FUNCTION F_VoltageToCurrentConvert : REAL
VAR_INPUT
	VoltageValue 	: REAL;
END_VAR
VAR
	Current			: REAL;
	Gain			: REAL := 3.1809;
	Offset			: REAL := -7.933;
END_VAR

Current := VoltageValue*Gain + Offset;

F_VoltageToCurrentConvert := Current;

END_FUNCTION

(* stored: Version 1.1.0.1, ProductVersion 3.1.4022.17
   POU F_VoltageToCurrentConvert: Id {4c259c44-8604-4beb-9049-3b9f090500ab}, SpecialFunc None *)
